FUNCTION_BLOCK FB_MAIN_CONV EXTENDS FB_STATION
VAR_INPUT
	fbAxis:REFERENCE TO FB_Axis;
END_VAR
VAR_OUTPUT
END_VAR
VAR
	bMOVE:BOOL :=FALSE;
	tNext: TON;
	tDelay: TON;
	bDELAY: BOOL:=FALSE;
	counter: INT;
	counter1: INT;
	bTest: INT;
	bSTARTUP: BOOL;
	total_length: INT;
	cart_space: INT;
	inc: INT;
	state: INT;
	temp: INT;
END_VAR

FOR counter:=1 TO num_of_carts BY 1 DO
	fbCART[counter]();
END_FOR;

IF NOT bFirstRun THEN
	A_set_cart_spaces();
	A_SETUP();
	bFirstRun:=TRUE;
END_IF



tDelay(IN:=bDELAY);
tNext(IN:=bMOVE , PT:=T#1S , Q=> , ET=> );

CASE eMAIN_CONVAYOR_STATE OF
	E_CONVAYOR_STATE.homing:
		bHomed:=TRUE;
		eMAIN_CONVAYOR_STATE:=E_CONVAYOR_STATE.idle;
		fbAxis.bEnable:=TRUE;
		fbAxis.bHalt:=FALSE;
		bDELAY:=FALSE;
		fbAxis.bSetPosition:=FALSE;
		fbAxis.bReset:=FALSE;
	
	E_CONVAYOR_STATE.uninit:
		IF NOT  bHomed THEN
			eMAIN_CONVAYOR_STATE:=E_CONVAYOR_STATE.homing;
		ELSE
			eMAIN_CONVAYOR_STATE:=E_CONVAYOR_STATE.idle;	
		END_IF
		fbAxis.bDo_Step_FW:=FALSE;
		fbAxis.bMoveRel:=FALSE;
		fbAxis.stepFW_state:=0;
		fbAxis.bHalt:=FALSE;
		fbAxis.bReset:=FALSE;
		
	E_CONVAYOR_STATE.idle:
		//
		
	E_CONVAYOR_STATE.do_move: // start motion
		IF NOT fbAxis.bBusy  AND NOT fbAxis.bError THEN
			fbAxis.rPos:=0;	
			fbAxis.bSetPosition:=TRUE;	 
			A_CARTS_STEP();
			fbAxis.bDo_Step_FW:=TRUE;
			eMAIN_CONVAYOR_STATE:=E_CONVAYOR_STATE.st1;
		END_IF
		
	E_CONVAYOR_STATE.st1:
		IF fbAxis.rActPos < 200 THEN
			eMAIN_CONVAYOR_STATE:=E_CONVAYOR_STATE.st2;	
			fbAxis.bSetPosition:=FALSE;
		END_IF
		
	E_CONVAYOR_STATE.st2:
		IF fbAxis.rActPos > (fbAxis.rStep/2)	THEN
			A_CARTS_STEP();	
			eMAIN_CONVAYOR_STATE:=E_CONVAYOR_STATE.st3;
		END_IF


	E_CONVAYOR_STATE.st3:
		IF fbAxis.bInPos THEN
			eMAIN_CONVAYOR_STATE:=E_CONVAYOR_STATE.done;
		END_IF
		
	E_CONVAYOR_STATE.done:
		//...
	
	E_CONVAYOR_STATE.pause:
	//
	
	E_CONVAYOR_STATE.estop:
		fbAxis.stepFW_state:=0;
		fbAxis.bHalt:=TRUE;
		fbAxis.bReset:=TRUE;
		bHomed:=FALSE;
	//...
	
	
END_CASE

ACTION A_CARTS_STEP:
FOR counter1:=1 TO num_of_carts BY 1 DO
	fbCART[counter1].A_STEP();
END_FOR;

bTest:= NOT bTest;
END_ACTION

ACTION A_set_cart_spaces:
 total_length := (conv_height*2)+(conv_length*2);
cart_space := total_length /((num_of_carts*2));
inc:=1;
posArrX[inc]:= 0+X_OFFSET;
posArrY[inc]:= 0+(conv_height/2)+Y_OFFSET;



WHILE state = 0 DO    //left1
	IF posArrY[inc]-cart_space < Y_OFFSET THEN
		temp :=cart_space - (posArrY[inc]-Y_OFFSET);
		posArrX[inc+1]:= temp+X_OFFSET;
		posArrY[inc+1]:= 0+Y_OFFSET;
		state:=1;
	ELSE
		posArrX[inc+1]:= 0+X_OFFSET;
		posArrY[inc+1]:=posArrY[inc]- cart_space;
		inc :=inc+1;
	END_IF
END_WHILE
inc := inc+1;

WHILE state = 1 DO // top
	IF posArrX[inc]+cart_space > (X_OFFSET+conv_length) THEN
		temp :=cart_space - ((X_OFFSET+conv_length)-posArrX[inc]);
		posArrX[inc+1]:= conv_length+X_OFFSET;
		posArrY[inc+1]:= temp+Y_OFFSET;
		state:=2;
	ELSE
		posArrX[inc+1]:= posArrX[inc]+cart_space;
		posArrY[inc+1]:=Y_OFFSET;
		inc :=inc+1;
	END_IF
END_WHILE
inc :=inc+1;	

WHILE state = 2 DO // right
	IF posArrY[inc]+cart_space > (Y_OFFSET+conv_height) THEN
		temp :=cart_space - ((Y_OFFSET+conv_height)-posArrY[inc]);
		posArrX[inc+1]:= (conv_length+X_OFFSET)-temp;
		posArrY[inc+1]:= 0+Y_OFFSET+conv_height;
		state:=3;
	ELSE
		posArrX[inc+1]:= 0+X_OFFSET+conv_length;
		posArrY[inc+1]:=posArrY[inc]+ cart_space;
		inc :=inc+1;
	END_IF	
END_WHILE
inc :=inc+1;	

WHILE state = 3 DO //bottom
	IF  posArrX[inc]-cart_space < X_OFFSET THEN
		temp :=cart_space - (posArrX[inc]-X_OFFSET);
		posArrX[inc+1]:= X_OFFSET;
		posArrY[inc+1]:= Y_OFFSET+ conv_height-temp;
		state:=4;
	ELSE
		posArrX[inc+1]:= posArrX[inc]-cart_space;
		posArrY[inc+1]:=Y_OFFSET+conv_height;
		inc :=inc+1;
		
	END_IF
END_WHILE

IF inc > 34 THEN
	RETURN;
END_IF


inc :=inc+1;

WHILE state = 4 DO    //left2
	IF posArrY[inc]-cart_space < ((conv_height/2)+Y_OFFSET) THEN
		state:=5;
	ELSE
		posArrX[inc+1]:= 0+X_OFFSET;
		posArrY[inc+1]:=posArrY[inc]- cart_space;
		inc :=inc+1;
		
	END_IF
END_WHILE
END_ACTION

ACTION A_SETUP:
bSTARTUP:=TRUE;
	fbCART[1].stCART.position:=1;
	fbCART[1].stCART.color:=1;
	fbCART[1].stCART.nNAME:=INT_TO_STRING(1001);
	fbCART[1].stCART.posX:=posArrX[1];
	fbCART[1].stCART.posY:=posArrY[1];
		
	FOR counter:=1 TO (num_of_carts-1) BY 1 DO
		fbCART[counter+1].stCART.position:=37-((counter*2));
		fbCART[counter+1].stCART.color:=1;
		fbCART[counter+1].stCART.nNAME:=INT_TO_STRING(1000+counter+1);
		fbCART[counter+1].stCART.posX:=posArrX[37-((counter*2))];
		fbCART[counter+1].stCART.posY:=posArrY[37-((counter*2))];
	END_FOR;
END_ACTION

END_FUNCTION_BLOCK

(* stored: Version 1.1.0.1, ProductVersion 3.1.4024.12
   POU FB_MAIN_CONV: Id {71cfab58-087d-476c-851d-edc288f639d5}, SpecialFunc None
   Action A_CARTS_STEP: Id {f1cd68c8-1db3-44d5-945e-848910b1fd9a}
   Action A_set_cart_spaces: Id {7785daa4-c212-4f07-a161-d0b471ee798f}
   Action A_SETUP: Id {20c6d030-312a-4e4f-82b8-3645da995266} *)
